Staubli VAL3: start.pgx

program start()
  local num l_nMean
  local num l_nMedian
  local num l_nVariance
  local num l_nStandardDeviation
  local num l_nGeoMean
  local num l_nRes
begin

  nInput[0] = 2
  nInput[1] = 1
  nInput[2] = 6
  nInput[3] = 5
  nInput[4] = 2
  nInput[5] = 4
  nInput[6] = 1
  nInput[7] = 7

  call getMean(nInput, l_nRes)
  ? "Mittelwert: " + toString(".4", l_nRes)

  call getMedian(nInput, l_nRes)
  ? "Median: " + toString(".4", l_nRes)

  call getVariance(nInput, l_nRes)
  ? "Varianz: " + toString(".4", l_nRes)

  call getStandardDeviation(nInput, l_nRes)
  ? "Std. Deviation: " + toString(".4", l_nRes)

  call getGeometricMean(nInput, l_nRes)
  ? "Geom. Mean: " + toString(".4", l_nRes)

  call getHarmonicMean(nInput, l_nRes)
  ? "Harm. Mean: " + toString(".4", l_nRes)
end
